# EPICS StreamDevice protocol: epics_installer_v1.0/option/serialTest_RAON_20220420/db/ACP40.proto
ReplyTimeout = 200;
InTerminator = CR;

# No outTerminator because we need to send ENQ clean or RS485 will mess up the reply.

#address = ESC "0\$1"; # for RS485

#handshake { wait 10; in ACK; out ENQ; wait 10; }

set2nominalspeed
{
    out "#\$1NSP" CR;
    in "#\$1,ok";
}

set_onoff
{
    out "#\$1%{ACPOFF|ACPON}" CR;
    in  "#\$1,ok";
}

read_status
{
    out "#\$1STA" CR;
    in "#\$1,"
       "%(\$2:STATUS.A)d,"
       "%(\$2:FAULT.A)d,"
       "%(\$2:ALERT.A)d,"
       "%(\$2:PUMP_ROTATION_SPEED.A)d,"
       "%(\$2:MOTOR_POWER.A)d,"
       "%(\$2:RESERVED.A)d,"
       "%(\$2:FREQUENCY_CONVERTER_TEMP.A)d,"
       "%(\$2:RESERVER.A)d,"
       "%(\$2:PUMP_OPERATING_TIME.A)d";
}

read_address
{
    out "#???ADR" CR;
    in "#%d,ok";
}

set_address
{
    out "#\$1ADR%d" CR;
    in "#%d,ok";
}
